Staubli VAL3: blink.pgx

public program blink(string x_sDioName, num x_nInterval, dio x_dDio)
begin

  //blink the output x_dDio with period x_nInterval

  if taskStatus("blink_"+x_sDioName)==-1
    taskCreate "blink_"+x_sDioName,10,exeBlink(x_dDio,x_nInterval)
    wait(taskStatus("blink_"+x_sDioName)==1)
  else
    //logMsg("libSignals/blink->can't create the blink task")
  endIf


end
